# EPICS substitutions: iocBoot/ioc13Mjolnir/pid_slow.substitutions
file "$(STD)/db/pid_control.db"
{
pattern
{P,            PID,        INP,           OUT,         LOPR,  HOPR,  DRVL,  DRVH,  PREC,   KP,  KI,   KD,  SCAN}
{13MNIR:,      PID1,   13ETC_1:Ti0,  13MNIR:E1608:Ao1,   0,    10,     0,    10,     3,    1.2,  1.,   0.,  ".1 second"}
}
